TYPE Python_Kamera_Daten_Status :
STRUCT
	
	 Busy						:BOOL;
	 IsDone						:BOOL;
	 PictureValid				:BOOL;
	 Active						:BOOL; 
 
END_STRUCT
END_TYPE

(* stored: Version 1.1.0.1, ProductVersion 3.1.4024.12
   DUT Python_Kamera_Daten_Status: Id {9490680c-a91c-42be-bd85-c782db2671ec} *)
